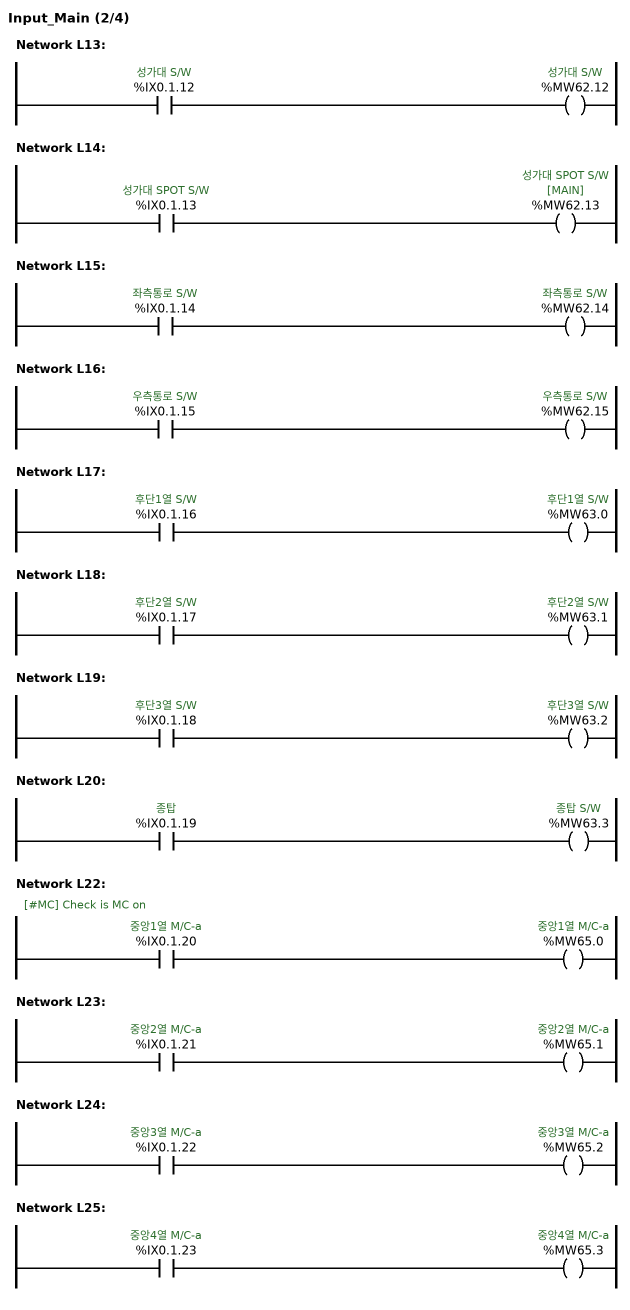
(* [picture p24: Input_Main rungs L13-L25] *)
(* Rung L13 *)
%MW62.12 := %IX0.1.12;
(* Rung L14 *)
%MW62.13 := %IX0.1.13;
(* Rung L15 *)
%MW62.14 := %IX0.1.14;
(* Rung L16 *)
%MW62.15 := %IX0.1.15;
(* Rung L17 *)
%MW63.0 := %IX0.1.16;
(* Rung L18 *)
%MW63.1 := %IX0.1.17;
(* Rung L19 *)
%MW63.2 := %IX0.1.18;
(* Rung L20 *)
%MW63.3 := %IX0.1.19;
(* [#MC] Check is MC on *)
(* Rung L22 *)
%MW65.0 := %IX0.1.20;
(* Rung L23 *)
%MW65.1 := %IX0.1.21;
(* Rung L24 *)
%MW65.2 := %IX0.1.22;
(* Rung L25 *)
%MW65.3 := %IX0.1.23;

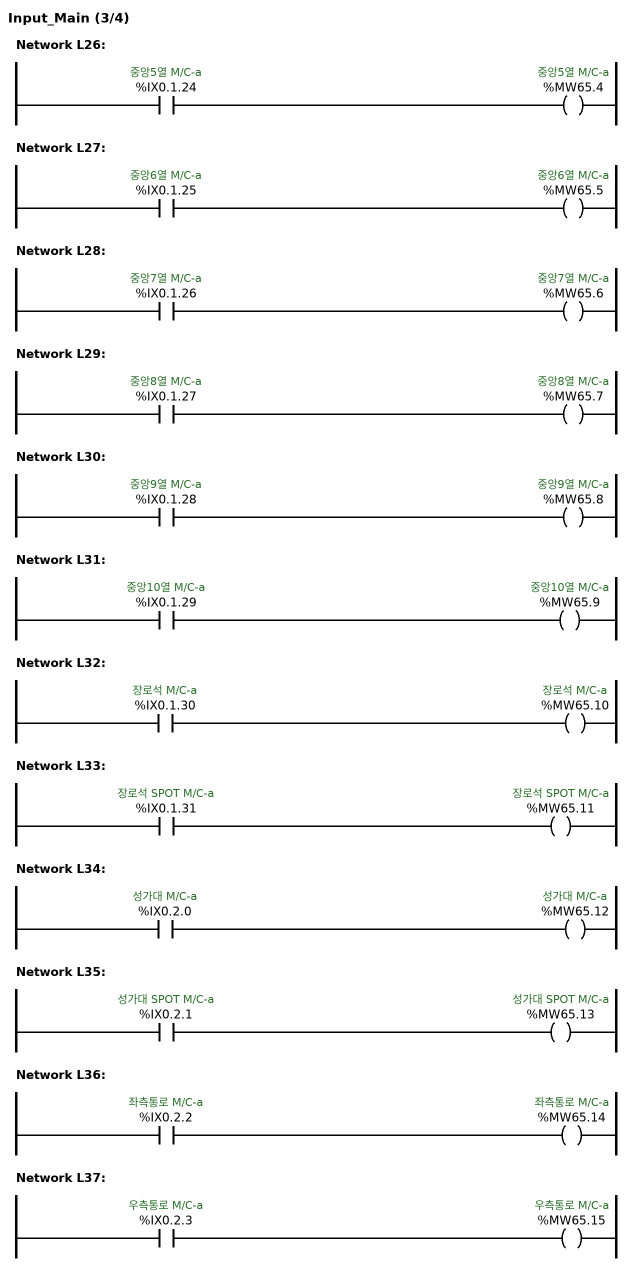
(* Rung L26 *)
%MW65.4 := %IX0.1.24;
(* Rung L27 *)
%MW65.5 := %IX0.1.25;
(* Rung L28 *)
%MW65.6 := %IX0.1.26;
(* Rung L29 *)
%MW65.7 := %IX0.1.27;
(* Rung L30 *)
%MW65.8 := %IX0.1.28;
(* Rung L31 *)
%MW65.9 := %IX0.1.29;
(* Rung L32 *)
%MW65.10 := %IX0.1.30;
(* Rung L33 *)
%MW65.11 := %IX0.1.31;
(* Rung L34 *)
%MW65.12 := %IX0.2.0;
(* Rung L35 *)
%MW65.13 := %IX0.2.1;
(* Rung L36 *)
%MW65.14 := %IX0.2.2;
(* Rung L37 *)
%MW65.15 := %IX0.2.3;

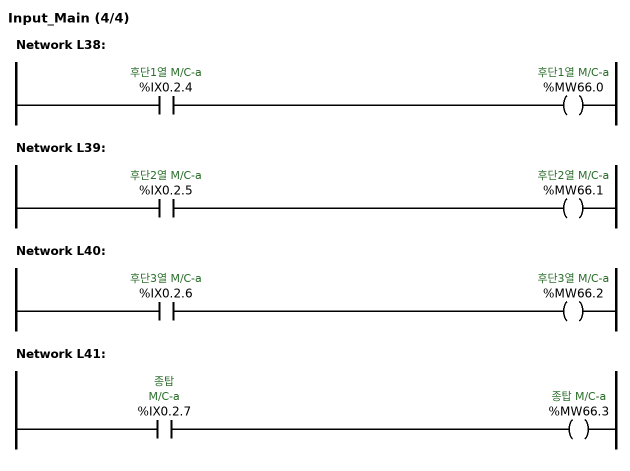
(* Rung L38 *)
%MW66.0 := %IX0.2.4;
(* Rung L39 *)
%MW66.1 := %IX0.2.5;
(* Rung L40 *)
%MW66.2 := %IX0.2.6;
(* Rung L41 *)
%MW66.3 := %IX0.2.7;
END_PROGRAM

PROGRAM Output-Main (* task: 스캔 프로그램 *)

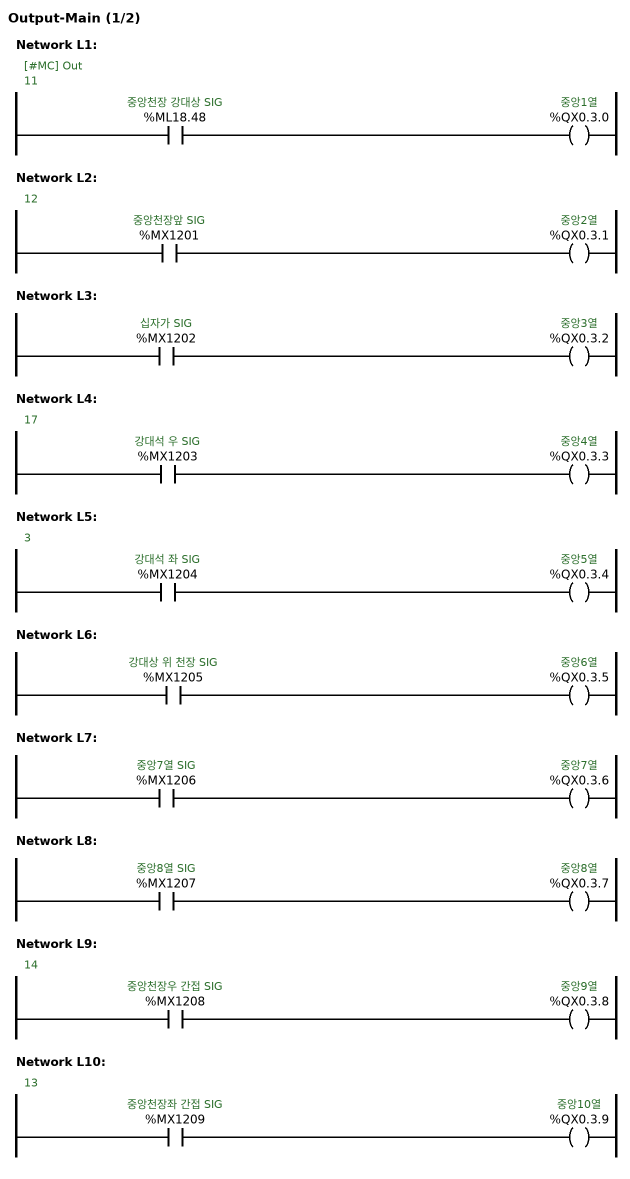
(* [#MC] Out *)
(* Rung L1 *)
%QX0.3.0 := %ML18.48;
(* 11 *)
(* Rung L2 *)
%QX0.3.1 := %MX1201;
(* 12 *)
(* Rung L3 *)
%QX0.3.2 := %MX1202;
(* Rung L4 *)
%QX0.3.3 := %MX1203;
(* 17 *)
(* Rung L5 *)
%QX0.3.4 := %MX1204;
(* 3 *)
(* Rung L6 *)
%QX0.3.5 := %MX1205;
(* Rung L7 *)
%QX0.3.6 := %MX1206;
(* Rung L8 *)
%QX0.3.7 := %MX1207;
(* Rung L9 *)
%QX0.3.8 := %MX1208;
(* 14 *)
(* Rung L10 *)
%QX0.3.9 := %MX1209;
(* 13 *)

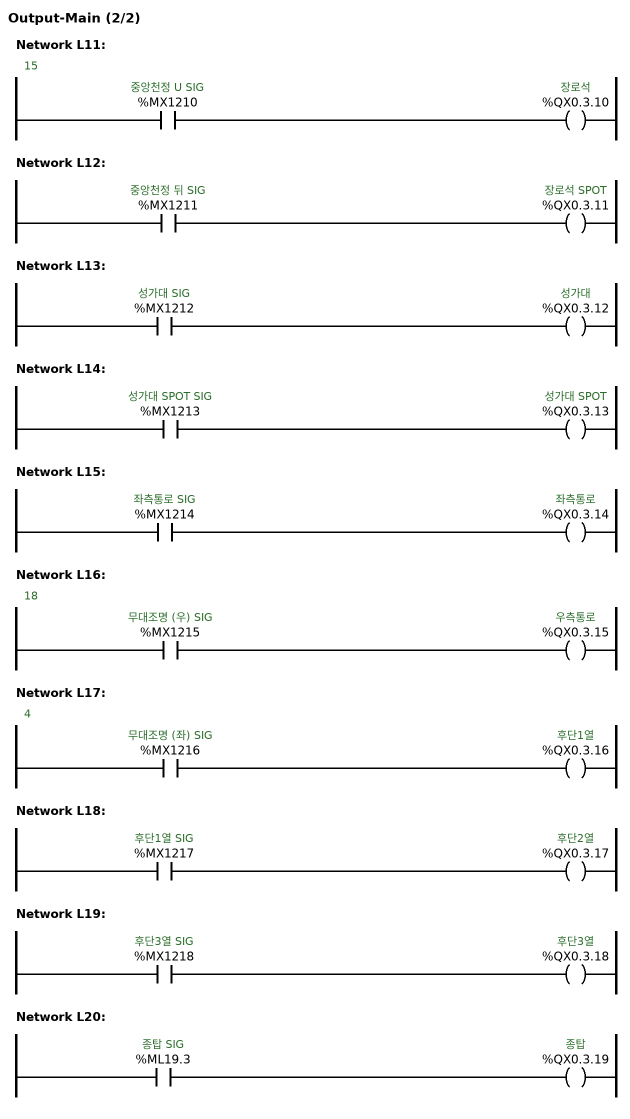
(* Rung L11 *)
%QX0.3.10 := %MX1210;
(* 15 *)
(* Rung L12 *)
%QX0.3.11 := %MX1211;
(* Rung L13 *)
%QX0.3.12 := %MX1212;
(* Rung L14 *)
%QX0.3.13 := %MX1213;
(* Rung L15 *)
%QX0.3.14 := %MX1214;
(* Rung L16 *)
%QX0.3.15 := %MX1215;
(* 18 *)
(* Rung L17 *)
%QX0.3.16 := %MX1216;
(* 4 *)
(* Rung L18 *)
%QX0.3.17 := %MX1217;
(* Rung L19 *)
%QX0.3.18 := %MX1218;
(* Rung L20 *)
%QX0.3.19 := %ML19.3;
END_PROGRAM

PROGRAM Alarm_Remote (* task: 스캔 프로그램 *)
VAR
    BUZZER : BOOL; (* BUZZER / SIG *)
    BZ_STOP : BOOL;
    FF : FF;
    INST : FF;
    INST1 : FF;
    INST2 : TON;
    INST9 : TMR_FLK;
END_VAR
VAR
    _p1 : BOOL;
    _t2 : BOOL;
END_VAR

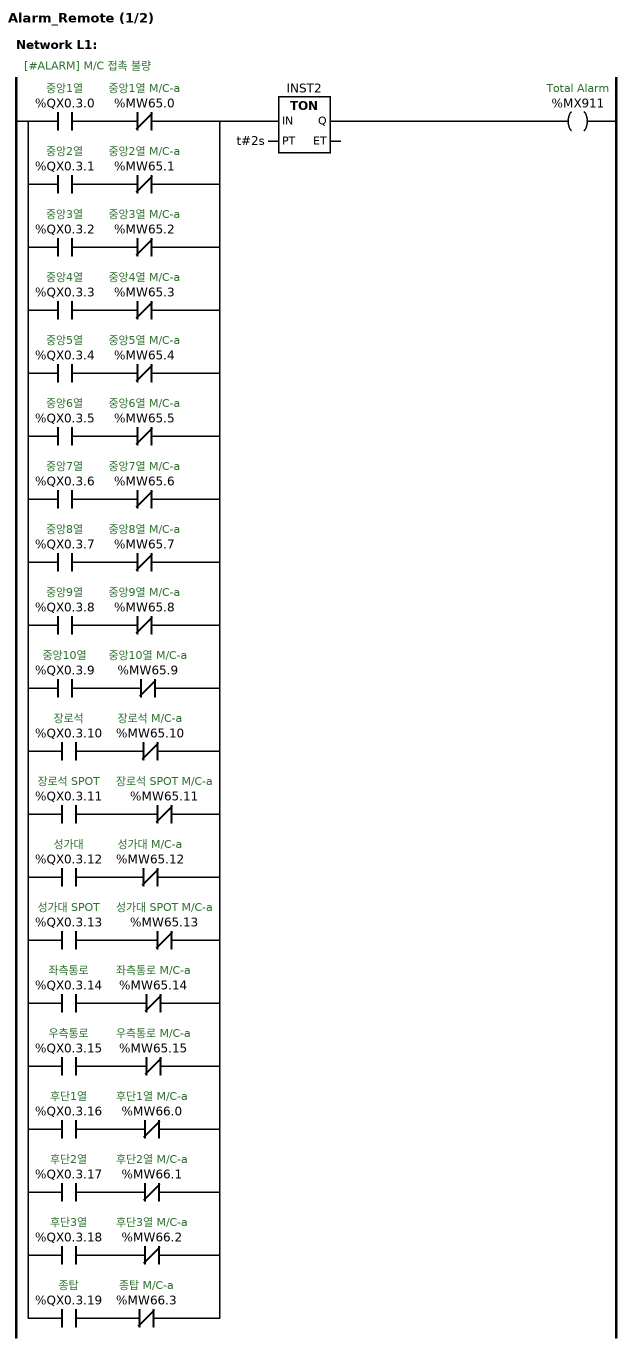
(* [#ALARM] M/C 접촉 불량 *)
(* Rung L1 *)
INST2(IN := (%QX0.3.0 AND NOT %MW65.0) OR (%QX0.3.1 AND NOT %MW65.1) OR (%QX0.3.2 AND NOT %MW65.2) OR (%QX0.3.3 AND NOT %MW65.3) OR (%QX0.3.4 AND NOT %MW65.4) OR (%QX0.3.5 AND NOT %MW65.5) OR (%QX0.3.6 AND NOT %MW65.6) OR (%QX0.3.7 AND NOT %MW65.7) OR (%QX0.3.8 AND NOT %MW65.8) OR (%QX0.3.9 AND NOT %MW65.9) OR (%QX0.3.10 AND NOT %MW65.10) OR (%QX0.3.11 AND NOT %MW65.11) OR (%QX0.3.12 AND NOT %MW65.12) OR (%QX0.3.13 AND NOT %MW65.13) OR (%QX0.3.14 AND NOT %MW65.14) OR (%QX0.3.15 AND NOT %MW65.15) OR (%QX0.3.16 AND NOT %MW66.0) OR (%QX0.3.17 AND NOT %MW66.1) OR (%QX0.3.18 AND NOT %MW66.2) OR (%QX0.3.19 AND NOT %MW66.3), PT := t#2s);
%MX911 := INST2.Q;

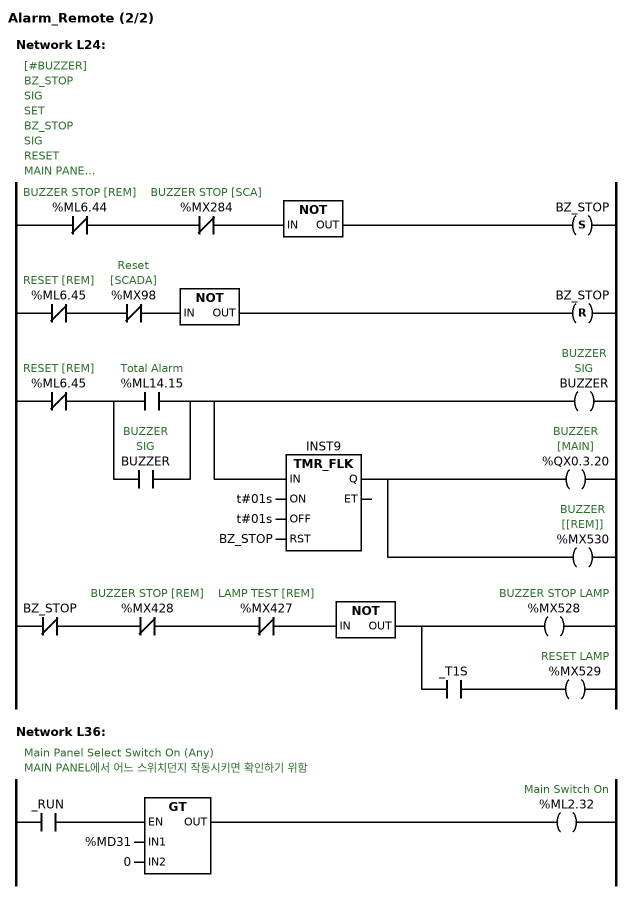
(* [#BUZZER] *)
(* Rung L24 *)
IF NOT (NOT %ML6.44 AND NOT %MX284) THEN BZ_STOP := TRUE; END_IF;
IF NOT (NOT %ML6.45 AND NOT %MX98) THEN BZ_STOP := FALSE; END_IF;
_p1 := NOT %ML6.45 AND (%ML14.15 OR BUZZER);
BUZZER := _p1;
INST9(IN := _p1, ON := t#01s, OFF := t#01s, RST := BZ_STOP);
%QX0.3.20 := INST9.Q;
%MX530 := INST9.Q;
%MX528 := NOT (NOT BZ_STOP AND NOT %MX428 AND NOT %MX427);
%MX529 := (NOT (NOT BZ_STOP AND NOT %MX428 AND NOT %MX427)) AND _T1S;
(* BZ_STOP / SIG / SET *)
(* BZ_STOP / SIG / RESET *)
(* MAIN PANEL / BUZZER / OUTPUT *)
(* [REM] PANEL / BUZZER / OUTPUT *)
(* Main Panel Select Switch On (Any) *)
(* Rung L36 *)
IF _RUN THEN _t2 := %MD31 > 0; END_IF;
%ML2.32 := _t2;
(* MAIN PANEL에서 어느 스위치던지 작동시키면 확인하기 위함 *)
END_PROGRAM